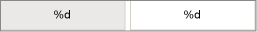
VISUALIZATION VISU_ConfigDINTEntry  // 257x32
VAR_IN_OUT
    active : DINT;
    editable : DINT;
END_VAR
    Textfield (0,0 125x30), "%d", text variable: active, input disabled if: TRUE
    Textfield (130,0 125x30), "%d", text variable: editable, colour toggle: editable <> active
        OnMouseClick: write the text variable via Default
END_VISUALIZATION

(* stored: Version 1.1.0.1, ProductVersion 3.1.4018.5
   Visu VISU_ConfigDINTEntry: Id {10210b98-09c2-49ee-a0bd-489e18e659a8} *)
